FUNCTION_BLOCK FB_Coordinador_SFC
VAR_INPUT
END_VAR
VAR_OUTPUT
END_VAR
VAR
END_VAR

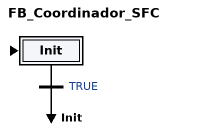
INITIAL_STEP Init:
END_STEP
TRANSITION FROM Init TO Init
    := TRUE;
END_TRANSITION

END_FUNCTION_BLOCK

(* stored: Version 1.1.0.1, ProductVersion 3.1.4024.12
   POU FB_Coordinador_SFC: Id {b557f5bf-c223-426b-b7fc-e7c2f78d1825}, SpecialFunc None *)
